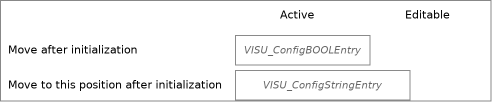
VISUALIZATION VISU_M3Config_General  // 492x102
VAR_IN_OUT
	active : M3Config;
	editable : M3Config;
END_VAR
    Label (235,5 125x20), "Active"
    Label (365,5 125x20), "Editable"
    Label (5,70 230x30), "Move to this position after initialization"
    Frame (235,70 175x30)
        shows VISU_ConfigStringEntry(active := active.moveAfterInitializationPosition, editable := editable.moveAfterInitializationPosition)
    Label (5,35 215x30), "Move after initialization"
    Frame (235,35 135x30)
        shows VISU_ConfigBOOLEntry(active := active.moveAfterInitialization, editable := editable.moveAfterInitialization)
END_VISUALIZATION

(* stored: Version 1.1.0.1, ProductVersion 3.1.4019.2
   Visu VISU_M3Config_General: Id {cb8dec5b-adc5-4d3a-b25a-5610f797d777} *)
